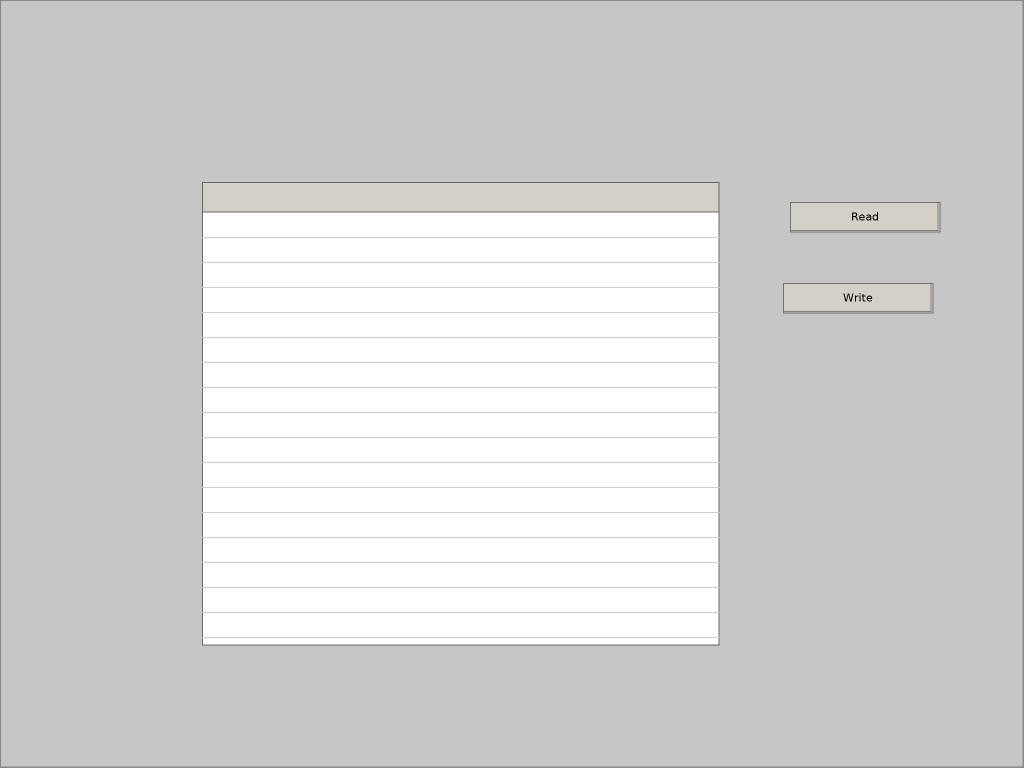
VISUALIZATION MaS_030_MenuScreen  // 1024x768
    Frame (0,0 1024x768)
        shows Tmp_000_Template(header := gHMIData.hmiHeader)
    Table (202,182 517x463), data array: MachineSettings.Setting
        p1420305297: MachineSettings.varSelectedColumn
        p4052804203: MachineSettings.varSelectedColumnValid
        p1137915858: MachineSettings.varSelectedRow
        p1822360349: MachineSettings.varSelectedRowValid
        p2232123230: MachineSettings.Setting[INDEX].TextName
        p511219082: MachineSettings.Setting[INDEX].Setting
    Button (790,202 150x30), "Read"
        tap MachineSettings.btnRead
    Button (783,283 150x30), "Write"
        tap MachineSettings.btnWrite
END_VISUALIZATION

(* stored: Version 1.1.0.1, ProductVersion 3.1.4024.11
   Visu MaS_030_MenuScreen: Id {44f1c459-314b-01ad-1879-0976785968a8} *)
